FUNCTION_BLOCK FastCounter EXTENDS TcoCore.TcoTask
VAR
	Counter : INT;	
	_counterProgressCheck :INT;
	_await : fbAwait;
END_VAR

IF Execute() THEN 
		

	IF _await.Delay(T#50MS) THEN
		Counter := Counter +1;
		_counterProgressCheck := Counter;
	END_IF
	
ThrowWhen(_counterProgressCheck > Counter);
	DoneWhen(Counter = 100);
	
END_IF

(*~
	<docu>
		<summary>
			Restores this instance to the Ready state. Can be called explicitly or from within one of the restore mechanisms.
			<para>
				See also <see cref="PlcDocu.TcoCore.TcoTask.AutoRestorable()"/>
			</para>
		</summary>			
	</docu>	
~*)
METHOD Restore : ITcoRestorable
SUPER^.Restore();
Counter := 0;
_counterProgressCheck:=0;
END_METHOD

END_FUNCTION_BLOCK

(* stored: Version 1.1.0.1, ProductVersion 3.1.4024.6
   POU FastCounter: Id {5b1cc310-97b4-0139-285e-18a442b4f3d9}, SpecialFunc None
   Method Restore: Id {424ed028-8a39-0c2e-3c50-32a912fad471} *)
